// SIMATIC S7-200 project (STEP 7-Micro/WIN), CPU 221 REL 01.10

SYMBOL_TABLE USUARIO1
Q1               I0.0     // Guardamotor protección motor (NA)
PG               I0.1     // Pulsador de paro general (NC)
P                I0.2     // Pulsador de paro fin de ciclo (NC)
PM               I0.3     // Pulsador de marcha
B1               I0.4     // Detector mezcla producto B
B2               I0.5     // Detector mezcla producto A
B3               I0.6     // Detector deposito vacío
M1               Q0.0     // Motor mezcladora
M2               Q0.1     // Cinta transportadora alimentación producto A
M3               Q0.2     // Cinta transportadora alimentación producto B
M4               Q0.3     // Cinta transportadora salida mezcla
H1               Q0.4     // Señalización intermitente mezcla ( Tiempo de
END_SYMBOL_TABLE

ORGANIZATION_BLOCK PRINCIPAL:OB1
TITLE=COMENTARIOS DEL PROGRAMA
BEGIN
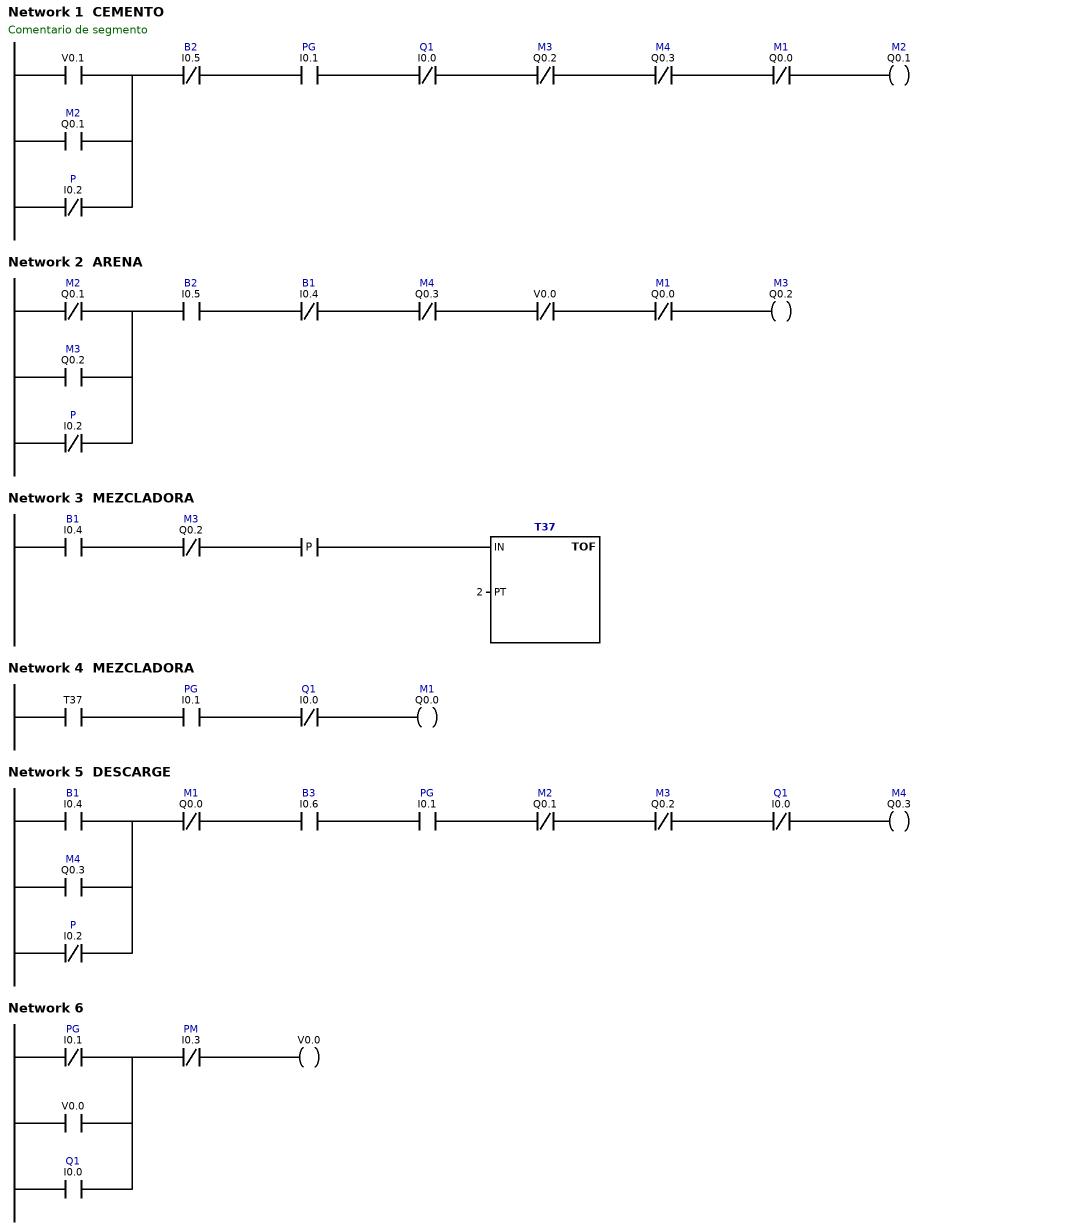
Network 1 // CEMENTO
// Comentario de segmento
LD     V0.1
O      M2:Q0.1
ON     P:I0.2
AN     B2:I0.5
A      PG:I0.1
AN     Q1:I0.0
AN     M3:Q0.2
AN     M4:Q0.3
AN     M1:Q0.0
=      M2:Q0.1
Network 2 // ARENA
LDN    M2:Q0.1
O      M3:Q0.2
ON     P:I0.2
A      B2:I0.5
AN     B1:I0.4
AN     M4:Q0.3
AN     V0.0
AN     M1:Q0.0
=      M3:Q0.2
Network 3 // MEZCLADORA
LD     B1:I0.4
AN     M3:Q0.2
EU
TOF    T37, 2
Network 4 // MEZCLADORA
LD     T37
A      PG:I0.1
AN     Q1:I0.0
=      M1:Q0.0
Network 5 // DESCARGE
LD     B1:I0.4
O      M4:Q0.3
ON     P:I0.2
AN     M1:Q0.0
A      B3:I0.6
A      PG:I0.1
AN     M2:Q0.1
AN     M3:Q0.2
AN     Q1:I0.0
=      M4:Q0.3
Network 6
LDN    PG:I0.1
O      V0.0
O      Q1:I0.0
AN     PM:I0.3
=      V0.0
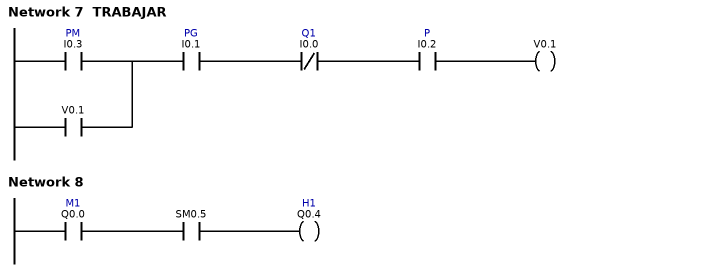
Network 7 // TRABAJAR
LD     PM:I0.3
O      V0.1
A      PG:I0.1
AN     Q1:I0.0
A      P:I0.2
=      V0.1
Network 8
LD     M1:Q0.0
A      SM0.5
=      H1:Q0.4
END_ORGANIZATION_BLOCK
